// TIA Portal V16 export
// export: Created 2021-09-22T12:44:53.8050822Z, ExportSetting WithDefaults, DisplayName Totally Integrated Automation Portal, DisplayVersion V16 Update 1, DisplayName TIA Portal Version Control Interface, DisplayVersion V16, DisplayName TIA Portal Openness, DisplayVersion V16, DisplayName SINAMICS Startdrive Advanced, DisplayVersion V16 Update 5, DisplayName SINAMICS Startdrive G130, G150, S120, S150, SINAMICS MV, S210, DisplayVersion V16 Update 5, DisplayName SINAMICS Startdrive G110M, G120, G120C, G120D, G120P, G115D, DisplayVersion V16 Update 5, DisplayName STEP 7 Professional, DisplayVersion V16, DisplayName STEP 7 Safety, DisplayVersion V16, DisplayName WinCC Professional, DisplayVersion V16
FUNCTION_BLOCK "FB_ChuteControl"   // FB4, LAD
{ S7_Optimized_Access := 'TRUE' }
VERSION : 0.1
// stored: AutoNumber true, IsIECCheckEnabled false, IsRetainMemResEnabled false, MemoryReserve 100, SetENOAutomatically false, UDAEnableTagReadback false
   VAR_INPUT
      Acil_OK : Bool;
      Otomatik : Bool;
      Hata_Reset : Bool;
   END_VAR
   VAR
      Yanaştırma : "FB549.Divert.Sorter.Basing";
      "FB548.Divert.Sorter.Chute_CN1_Divert1" { S7_SetPoint := 'True'} : "FB548.Divert.Sorter.Chute";
      "FB548.Divert.Sorter.Chute_CN2_Divert2" { S7_SetPoint := 'True'} : "FB548.Divert.Sorter.Chute";
      "FB548.Divert.Sorter.Chute_CN3_Divert3" { S7_SetPoint := 'True'} : "FB548.Divert.Sorter.Chute";
      "FB548.Divert.Sorter.Chute_CN4_Divert4" { S7_SetPoint := 'True'} : "FB548.Divert.Sorter.Chute";
      "FB548.Divert.Sorter.Chute_CN5_Divert5" { S7_SetPoint := 'True'} : "FB548.Divert.Sorter.Chute";
   END_VAR
   VAR_TEMP
      i : Int;
      j : Int;
   END_VAR
   VAR_TEMP   // added for the SCL form of the ladder/FBD networks
      _w1 : Bool;
   END_VAR
BEGIN

REGION Network 1: CN2 POS1065 Divert1
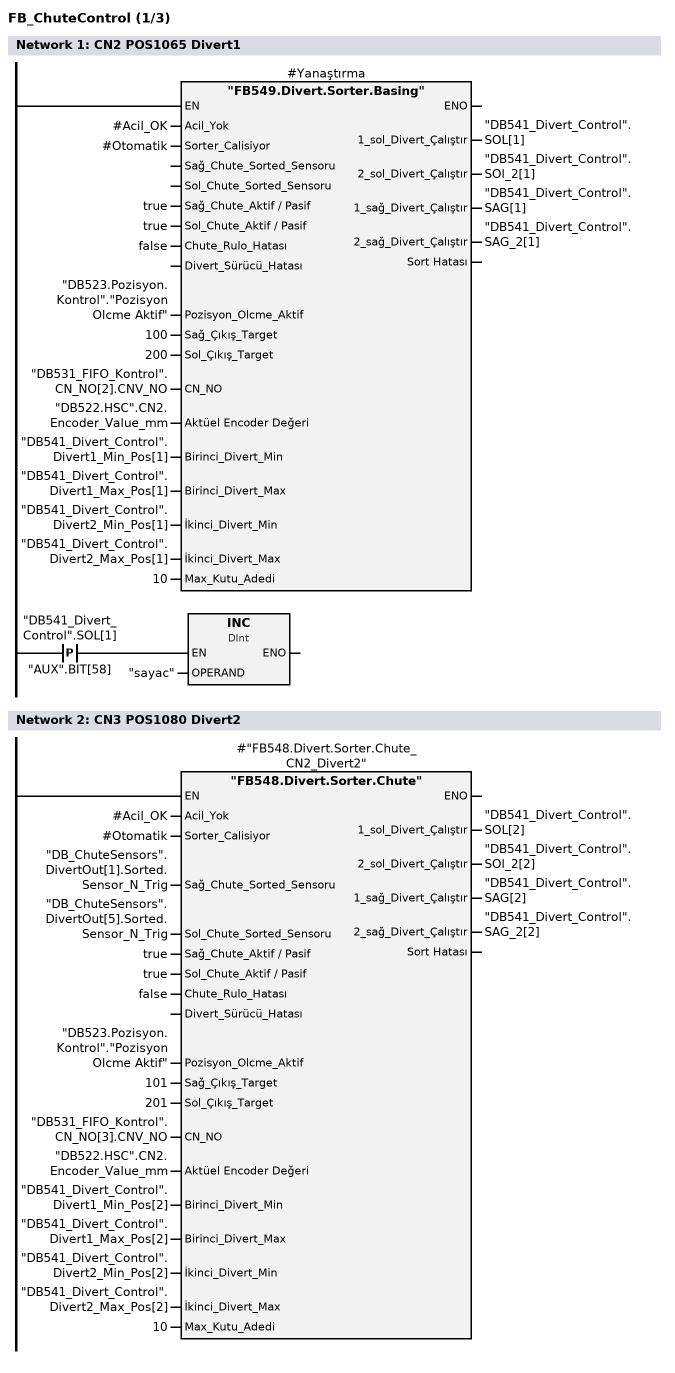
   RUNG wire#powerrail
      #Yanaştırma(Acil_Yok := #Acil_OK, Sorter_Calisiyor := #Otomatik, Sağ_Chute_Sorted_Sensoru :=, Sol_Chute_Sorted_Sensoru :=, "Sağ_Chute_Aktif / Pasif" := true, "Sol_Chute_Aktif / Pasif" := true, Chute_Rulo_Hatası := false, Divert_Sürücü_Hatası :=, Pozisyon_Olcme_Aktif := "DB523.Pozisyon.Kontrol"."Pozisyon Olcme Aktif", Sağ_Çıkış_Target := 100, Sol_Çıkış_Target := 200, CN_NO := "DB531_FIFO_Kontrol".CN_NO[2].CNV_NO, "Aktüel Encoder Değeri" := "DB522.HSC".CN2.Encoder_Value_mm, Birinci_Divert_Min := "DB541_Divert_Control".Divert1_Min_Pos[1], Birinci_Divert_Max := "DB541_Divert_Control".Divert1_Max_Pos[1], İkinci_Divert_Min := "DB541_Divert_Control".Divert2_Min_Pos[1], İkinci_Divert_Max := "DB541_Divert_Control".Divert2_Max_Pos[1], Max_Kutu_Adedi := 10, "1_sol_Divert_Çalıştır" => "DB541_Divert_Control".SOL[1], "2_sol_Divert_Çalıştır" => "DB541_Divert_Control".SOl_2[1], "1_sağ_Divert_Çalıştır" => "DB541_Divert_Control".SAG[1], "2_sağ_Divert_Çalıştır" => "DB541_Divert_Control".SAG_2[1], "Sort Hatası" =>)
   END_RUNG
   RUNG wire#powerrail
      P_Contact(operand := "DB541_Divert_Control".SOL[1], bit := "AUX".BIT[58])
      { S7_Templates := "DestType := DInt" } Inc( "sayac" )
   END_RUNG
   // the same network as SCL:
   #Yanaştırma(Acil_Yok := #Acil_OK,   // "FB549.Divert.Sorter.Basing"
               Sorter_Calisiyor := #Otomatik,
               "Sağ_Chute_Aktif / Pasif" := true,
               "Sol_Chute_Aktif / Pasif" := true,
               Chute_Rulo_Hatası := false,
               Pozisyon_Olcme_Aktif := "DB523.Pozisyon.Kontrol"."Pozisyon Olcme Aktif",
               Sağ_Çıkış_Target := 100,
               Sol_Çıkış_Target := 200,
               CN_NO := "DB531_FIFO_Kontrol".CN_NO[2].CNV_NO,
               "Aktüel Encoder Değeri" := "DB522.HSC".CN2.Encoder_Value_mm,
               Birinci_Divert_Min := "DB541_Divert_Control".Divert1_Min_Pos[1],
               Birinci_Divert_Max := "DB541_Divert_Control".Divert1_Max_Pos[1],
               İkinci_Divert_Min := "DB541_Divert_Control".Divert2_Min_Pos[1],
               İkinci_Divert_Max := "DB541_Divert_Control".Divert2_Max_Pos[1],
               Max_Kutu_Adedi := 10,
               "1_sol_Divert_Çalıştır" => "DB541_Divert_Control".SOL[1],
               "2_sol_Divert_Çalıştır" => "DB541_Divert_Control".SOl_2[1],
               "1_sağ_Divert_Çalıştır" => "DB541_Divert_Control".SAG[1],
               "2_sağ_Divert_Çalıştır" => "DB541_Divert_Control".SAG_2[1]);
   #_w1 := "DB541_Divert_Control".SOL[1] AND NOT "AUX".BIT[58];   // rising edge of "DB541_Divert_Control".SOL[1]
   "AUX".BIT[58] := "DB541_Divert_Control".SOL[1];
   IF #_w1 THEN "sayac" := "sayac" + 1; END_IF;
END_REGION

REGION Network 2: CN3 POS1080 Divert2
   RUNG wire#powerrail
      #"FB548.Divert.Sorter.Chute_CN2_Divert2"(Acil_Yok := #Acil_OK, Sorter_Calisiyor := #Otomatik, Sağ_Chute_Sorted_Sensoru := "DB_ChuteSensors".DivertOut[1].Sorted.Sensor_N_Trig, Sol_Chute_Sorted_Sensoru := "DB_ChuteSensors".DivertOut[5].Sorted.Sensor_N_Trig, "Sağ_Chute_Aktif / Pasif" := true, "Sol_Chute_Aktif / Pasif" := true, Chute_Rulo_Hatası := false, Divert_Sürücü_Hatası :=, Pozisyon_Olcme_Aktif := "DB523.Pozisyon.Kontrol"."Pozisyon Olcme Aktif", Sağ_Çıkış_Target := 101, Sol_Çıkış_Target := 201, CN_NO := "DB531_FIFO_Kontrol".CN_NO[3].CNV_NO, "Aktüel Encoder Değeri" := "DB522.HSC".CN2.Encoder_Value_mm, Birinci_Divert_Min := "DB541_Divert_Control".Divert1_Min_Pos[2], Birinci_Divert_Max := "DB541_Divert_Control".Divert1_Max_Pos[2], İkinci_Divert_Min := "DB541_Divert_Control".Divert2_Min_Pos[2], İkinci_Divert_Max := "DB541_Divert_Control".Divert2_Max_Pos[2], Max_Kutu_Adedi := 10, "1_sol_Divert_Çalıştır" => "DB541_Divert_Control".SOL[2], "2_sol_Divert_Çalıştır" => "DB541_Divert_Control".SOl_2[2], "1_sağ_Divert_Çalıştır" => "DB541_Divert_Control".SAG[2], "2_sağ_Divert_Çalıştır" => "DB541_Divert_Control".SAG_2[2], "Sort Hatası" =>)
   END_RUNG
   // the same network as SCL:
   #"FB548.Divert.Sorter.Chute_CN2_Divert2"(Acil_Yok := #Acil_OK,   // "FB548.Divert.Sorter.Chute"
                           Sorter_Calisiyor := #Otomatik,
                           Sağ_Chute_Sorted_Sensoru := "DB_ChuteSensors".DivertOut[1].Sorted.Sensor_N_Trig,
                           Sol_Chute_Sorted_Sensoru := "DB_ChuteSensors".DivertOut[5].Sorted.Sensor_N_Trig,
                           "Sağ_Chute_Aktif / Pasif" := true,
                           "Sol_Chute_Aktif / Pasif" := true,
                           Chute_Rulo_Hatası := false,
                           Pozisyon_Olcme_Aktif := "DB523.Pozisyon.Kontrol"."Pozisyon Olcme Aktif",
                           Sağ_Çıkış_Target := 101,
                           Sol_Çıkış_Target := 201,
                           CN_NO := "DB531_FIFO_Kontrol".CN_NO[3].CNV_NO,
                           "Aktüel Encoder Değeri" := "DB522.HSC".CN2.Encoder_Value_mm,
                           Birinci_Divert_Min := "DB541_Divert_Control".Divert1_Min_Pos[2],
                           Birinci_Divert_Max := "DB541_Divert_Control".Divert1_Max_Pos[2],
                           İkinci_Divert_Min := "DB541_Divert_Control".Divert2_Min_Pos[2],
                           İkinci_Divert_Max := "DB541_Divert_Control".Divert2_Max_Pos[2],
                           Max_Kutu_Adedi := 10,
                           "1_sol_Divert_Çalıştır" => "DB541_Divert_Control".SOL[2],
                           "2_sol_Divert_Çalıştır" => "DB541_Divert_Control".SOl_2[2],
                           "1_sağ_Divert_Çalıştır" => "DB541_Divert_Control".SAG[2],
                           "2_sağ_Divert_Çalıştır" => "DB541_Divert_Control".SAG_2[2]);
END_REGION

REGION Network 3 (SCL)


   IF "DB541_Divert_Control".SOL[2] THEN
       "DB541_Divert_Control".SOl_2[2] := TRUE;
   END_IF;

   IF "DB541_Divert_Control".SAG[2] THEN
       "DB541_Divert_Control".SAG_2[2] := TRUE;
   END_IF;
END_REGION

REGION Network 4: CN4 POS1190 Divert3
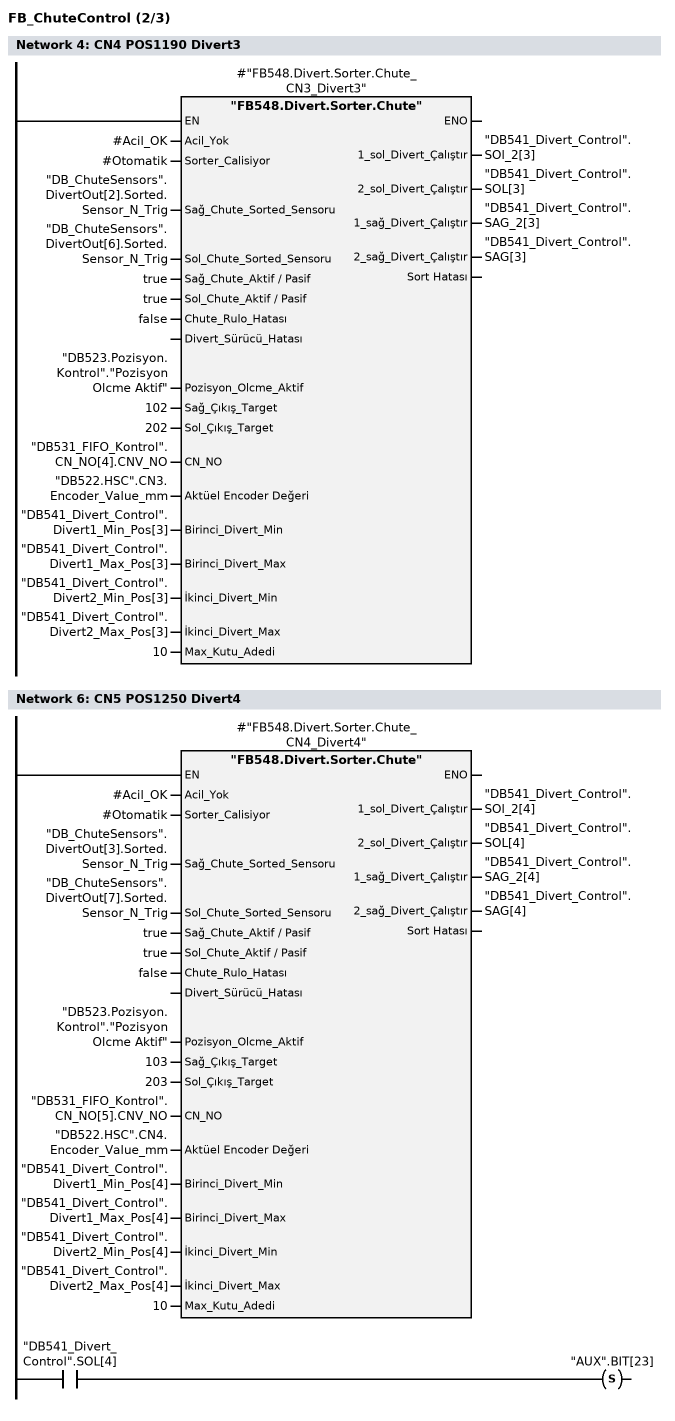
   RUNG wire#powerrail
      #"FB548.Divert.Sorter.Chute_CN3_Divert3"(Acil_Yok := #Acil_OK, Sorter_Calisiyor := #Otomatik, Sağ_Chute_Sorted_Sensoru := "DB_ChuteSensors".DivertOut[2].Sorted.Sensor_N_Trig, Sol_Chute_Sorted_Sensoru := "DB_ChuteSensors".DivertOut[6].Sorted.Sensor_N_Trig, "Sağ_Chute_Aktif / Pasif" := true, "Sol_Chute_Aktif / Pasif" := true, Chute_Rulo_Hatası := false, Divert_Sürücü_Hatası :=, Pozisyon_Olcme_Aktif := "DB523.Pozisyon.Kontrol"."Pozisyon Olcme Aktif", Sağ_Çıkış_Target := 102, Sol_Çıkış_Target := 202, CN_NO := "DB531_FIFO_Kontrol".CN_NO[4].CNV_NO, "Aktüel Encoder Değeri" := "DB522.HSC".CN3.Encoder_Value_mm, Birinci_Divert_Min := "DB541_Divert_Control".Divert1_Min_Pos[3], Birinci_Divert_Max := "DB541_Divert_Control".Divert1_Max_Pos[3], İkinci_Divert_Min := "DB541_Divert_Control".Divert2_Min_Pos[3], İkinci_Divert_Max := "DB541_Divert_Control".Divert2_Max_Pos[3], Max_Kutu_Adedi := 10, "1_sol_Divert_Çalıştır" => "DB541_Divert_Control".SOl_2[3], "2_sol_Divert_Çalıştır" => "DB541_Divert_Control".SOL[3], "1_sağ_Divert_Çalıştır" => "DB541_Divert_Control".SAG_2[3], "2_sağ_Divert_Çalıştır" => "DB541_Divert_Control".SAG[3], "Sort Hatası" =>)
   END_RUNG
   // the same network as SCL:
   #"FB548.Divert.Sorter.Chute_CN3_Divert3"(Acil_Yok := #Acil_OK,   // "FB548.Divert.Sorter.Chute"
                           Sorter_Calisiyor := #Otomatik,
                           Sağ_Chute_Sorted_Sensoru := "DB_ChuteSensors".DivertOut[2].Sorted.Sensor_N_Trig,
                           Sol_Chute_Sorted_Sensoru := "DB_ChuteSensors".DivertOut[6].Sorted.Sensor_N_Trig,
                           "Sağ_Chute_Aktif / Pasif" := true,
                           "Sol_Chute_Aktif / Pasif" := true,
                           Chute_Rulo_Hatası := false,
                           Pozisyon_Olcme_Aktif := "DB523.Pozisyon.Kontrol"."Pozisyon Olcme Aktif",
                           Sağ_Çıkış_Target := 102,
                           Sol_Çıkış_Target := 202,
                           CN_NO := "DB531_FIFO_Kontrol".CN_NO[4].CNV_NO,
                           "Aktüel Encoder Değeri" := "DB522.HSC".CN3.Encoder_Value_mm,
                           Birinci_Divert_Min := "DB541_Divert_Control".Divert1_Min_Pos[3],
                           Birinci_Divert_Max := "DB541_Divert_Control".Divert1_Max_Pos[3],
                           İkinci_Divert_Min := "DB541_Divert_Control".Divert2_Min_Pos[3],
                           İkinci_Divert_Max := "DB541_Divert_Control".Divert2_Max_Pos[3],
                           Max_Kutu_Adedi := 10,
                           "1_sol_Divert_Çalıştır" => "DB541_Divert_Control".SOl_2[3],
                           "2_sol_Divert_Çalıştır" => "DB541_Divert_Control".SOL[3],
                           "1_sağ_Divert_Çalıştır" => "DB541_Divert_Control".SAG_2[3],
                           "2_sağ_Divert_Çalıştır" => "DB541_Divert_Control".SAG[3]);
END_REGION

REGION Network 5 (SCL)


   IF "DB541_Divert_Control".SOl_2[3] THEN
       "DB541_Divert_Control".SOL[3] := TRUE;
   END_IF;

   IF "DB541_Divert_Control".SAG_2[3] THEN
       "DB541_Divert_Control".SAG[3] := TRUE;
   END_IF;
END_REGION

REGION Network 6: CN5 POS1250 Divert4
   RUNG wire#powerrail
      #"FB548.Divert.Sorter.Chute_CN4_Divert4"(Acil_Yok := #Acil_OK, Sorter_Calisiyor := #Otomatik, Sağ_Chute_Sorted_Sensoru := "DB_ChuteSensors".DivertOut[3].Sorted.Sensor_N_Trig, Sol_Chute_Sorted_Sensoru := "DB_ChuteSensors".DivertOut[7].Sorted.Sensor_N_Trig, "Sağ_Chute_Aktif / Pasif" := true, "Sol_Chute_Aktif / Pasif" := true, Chute_Rulo_Hatası := false, Divert_Sürücü_Hatası :=, Pozisyon_Olcme_Aktif := "DB523.Pozisyon.Kontrol"."Pozisyon Olcme Aktif", Sağ_Çıkış_Target := 103, Sol_Çıkış_Target := 203, CN_NO := "DB531_FIFO_Kontrol".CN_NO[5].CNV_NO, "Aktüel Encoder Değeri" := "DB522.HSC".CN4.Encoder_Value_mm, Birinci_Divert_Min := "DB541_Divert_Control".Divert1_Min_Pos[4], Birinci_Divert_Max := "DB541_Divert_Control".Divert1_Max_Pos[4], İkinci_Divert_Min := "DB541_Divert_Control".Divert2_Min_Pos[4], İkinci_Divert_Max := "DB541_Divert_Control".Divert2_Max_Pos[4], Max_Kutu_Adedi := 10, "1_sol_Divert_Çalıştır" => "DB541_Divert_Control".SOl_2[4], "2_sol_Divert_Çalıştır" => "DB541_Divert_Control".SOL[4], "1_sağ_Divert_Çalıştır" => "DB541_Divert_Control".SAG_2[4], "2_sağ_Divert_Çalıştır" => "DB541_Divert_Control".SAG[4], "Sort Hatası" =>)
   END_RUNG
   RUNG wire#powerrail
      Contact( "DB541_Divert_Control".SOL[4] )
      S_Coil( "AUX".BIT[23] )
   END_RUNG
   // the same network as SCL:
   #"FB548.Divert.Sorter.Chute_CN4_Divert4"(Acil_Yok := #Acil_OK,   // "FB548.Divert.Sorter.Chute"
                           Sorter_Calisiyor := #Otomatik,
                           Sağ_Chute_Sorted_Sensoru := "DB_ChuteSensors".DivertOut[3].Sorted.Sensor_N_Trig,
                           Sol_Chute_Sorted_Sensoru := "DB_ChuteSensors".DivertOut[7].Sorted.Sensor_N_Trig,
                           "Sağ_Chute_Aktif / Pasif" := true,
                           "Sol_Chute_Aktif / Pasif" := true,
                           Chute_Rulo_Hatası := false,
                           Pozisyon_Olcme_Aktif := "DB523.Pozisyon.Kontrol"."Pozisyon Olcme Aktif",
                           Sağ_Çıkış_Target := 103,
                           Sol_Çıkış_Target := 203,
                           CN_NO := "DB531_FIFO_Kontrol".CN_NO[5].CNV_NO,
                           "Aktüel Encoder Değeri" := "DB522.HSC".CN4.Encoder_Value_mm,
                           Birinci_Divert_Min := "DB541_Divert_Control".Divert1_Min_Pos[4],
                           Birinci_Divert_Max := "DB541_Divert_Control".Divert1_Max_Pos[4],
                           İkinci_Divert_Min := "DB541_Divert_Control".Divert2_Min_Pos[4],
                           İkinci_Divert_Max := "DB541_Divert_Control".Divert2_Max_Pos[4],
                           Max_Kutu_Adedi := 10,
                           "1_sol_Divert_Çalıştır" => "DB541_Divert_Control".SOl_2[4],
                           "2_sol_Divert_Çalıştır" => "DB541_Divert_Control".SOL[4],
                           "1_sağ_Divert_Çalıştır" => "DB541_Divert_Control".SAG_2[4],
                           "2_sağ_Divert_Çalıştır" => "DB541_Divert_Control".SAG[4]);
   IF "DB541_Divert_Control".SOL[4] THEN "AUX".BIT[23] := TRUE; END_IF;
END_REGION

REGION Network 7 (SCL)


   IF "DB541_Divert_Control".SOl_2[4] THEN
       "DB541_Divert_Control".SOL[4] := TRUE;
   END_IF;

   IF "DB541_Divert_Control".SAG_2[4] THEN
       "DB541_Divert_Control".SAG[4] := TRUE;
   END_IF;
END_REGION

REGION Network 8: CN6 POS1310 Divert5
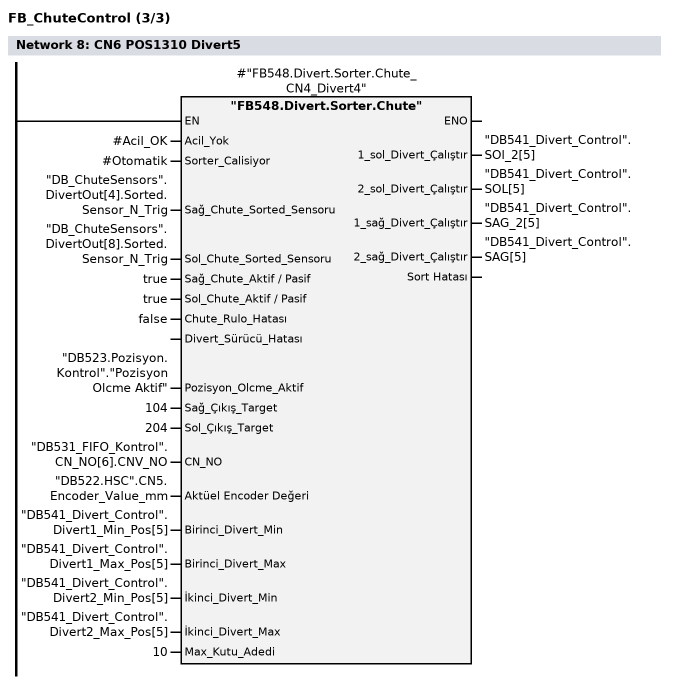
   RUNG wire#powerrail
      #"FB548.Divert.Sorter.Chute_CN4_Divert4"(Acil_Yok := #Acil_OK, Sorter_Calisiyor := #Otomatik, Sağ_Chute_Sorted_Sensoru := "DB_ChuteSensors".DivertOut[4].Sorted.Sensor_N_Trig, Sol_Chute_Sorted_Sensoru := "DB_ChuteSensors".DivertOut[8].Sorted.Sensor_N_Trig, "Sağ_Chute_Aktif / Pasif" := true, "Sol_Chute_Aktif / Pasif" := true, Chute_Rulo_Hatası := false, Divert_Sürücü_Hatası :=, Pozisyon_Olcme_Aktif := "DB523.Pozisyon.Kontrol"."Pozisyon Olcme Aktif", Sağ_Çıkış_Target := 104, Sol_Çıkış_Target := 204, CN_NO := "DB531_FIFO_Kontrol".CN_NO[6].CNV_NO, "Aktüel Encoder Değeri" := "DB522.HSC".CN5.Encoder_Value_mm, Birinci_Divert_Min := "DB541_Divert_Control".Divert1_Min_Pos[5], Birinci_Divert_Max := "DB541_Divert_Control".Divert1_Max_Pos[5], İkinci_Divert_Min := "DB541_Divert_Control".Divert2_Min_Pos[5], İkinci_Divert_Max := "DB541_Divert_Control".Divert2_Max_Pos[5], Max_Kutu_Adedi := 10, "1_sol_Divert_Çalıştır" => "DB541_Divert_Control".SOl_2[5], "2_sol_Divert_Çalıştır" => "DB541_Divert_Control".SOL[5], "1_sağ_Divert_Çalıştır" => "DB541_Divert_Control".SAG_2[5], "2_sağ_Divert_Çalıştır" => "DB541_Divert_Control".SAG[5], "Sort Hatası" =>)
   END_RUNG
   // the same network as SCL:
   #"FB548.Divert.Sorter.Chute_CN4_Divert4"(Acil_Yok := #Acil_OK,   // "FB548.Divert.Sorter.Chute"
                           Sorter_Calisiyor := #Otomatik,
                           Sağ_Chute_Sorted_Sensoru := "DB_ChuteSensors".DivertOut[4].Sorted.Sensor_N_Trig,
                           Sol_Chute_Sorted_Sensoru := "DB_ChuteSensors".DivertOut[8].Sorted.Sensor_N_Trig,
                           "Sağ_Chute_Aktif / Pasif" := true,
                           "Sol_Chute_Aktif / Pasif" := true,
                           Chute_Rulo_Hatası := false,
                           Pozisyon_Olcme_Aktif := "DB523.Pozisyon.Kontrol"."Pozisyon Olcme Aktif",
                           Sağ_Çıkış_Target := 104,
                           Sol_Çıkış_Target := 204,
                           CN_NO := "DB531_FIFO_Kontrol".CN_NO[6].CNV_NO,
                           "Aktüel Encoder Değeri" := "DB522.HSC".CN5.Encoder_Value_mm,
                           Birinci_Divert_Min := "DB541_Divert_Control".Divert1_Min_Pos[5],
                           Birinci_Divert_Max := "DB541_Divert_Control".Divert1_Max_Pos[5],
                           İkinci_Divert_Min := "DB541_Divert_Control".Divert2_Min_Pos[5],
                           İkinci_Divert_Max := "DB541_Divert_Control".Divert2_Max_Pos[5],
                           Max_Kutu_Adedi := 10,
                           "1_sol_Divert_Çalıştır" => "DB541_Divert_Control".SOl_2[5],
                           "2_sol_Divert_Çalıştır" => "DB541_Divert_Control".SOL[5],
                           "1_sağ_Divert_Çalıştır" => "DB541_Divert_Control".SAG_2[5],
                           "2_sağ_Divert_Çalıştır" => "DB541_Divert_Control".SAG[5]);
END_REGION

REGION Network 9 (SCL)


   IF "DB541_Divert_Control".SOl_2[5] THEN
       "DB541_Divert_Control".SOL[5] := TRUE;
   END_IF;

   IF "DB541_Divert_Control".SAG_2[5] THEN
       "DB541_Divert_Control".SAG[5] := TRUE;
   END_IF;
END_REGION
END_FUNCTION_BLOCK
